FUNCTION_BLOCK FB_SignalLight
VAR_INPUT
	eSafetyState	: E_SafetyState;
	eMachineState 	: E_MachineState;	
END_VAR
VAR_OUTPUT
END_VAR
VAR
	//Blink
	tmrBlink : TON;
	nStateBlink : USINT;
	bBlink	: BOOL;
	
	//Ausgänge für LEDs
	bRed 	AT %Q* : BOOL;
	bYellow AT %Q* : BOOL;
	bGreen	AT %Q* : BOOL;
END_VAR

A_Blink();
IF eSafetyState = E_SafetyState.EmergencyStopPressed THEN
	//rot blinkend
	bRed := TRUE AND bBlink;
	bYellow := FALSE;
	bGreen := FALSE;
	RETURN;
END_IF

CASE eMachineState OF
	E_MachineState.MACHINESTATE_Active, E_MachineState.MACHINESTATE_Running:
		bRed := FALSE;
		bYellow := FALSE;
		bGreen := TRUE;
	E_MachineState.MACHINESTATE_Error:
		bRed := TRUE;
		bYellow := FALSE;
		bGreen := FALSE;		
	E_MachineState.MACHINESTATE_Idle:
		bRed := FALSE;
		bGreen := FALSE;
		IF eSafetyState = E_SafetyState.Locked THEN
			bYellow := TRUE;
		ELSE
			bYellow := TRUE AND bBlink;
		END_IF
	ELSE
		bRed := FALSE;
		bYellow := FALSE;
		bGreen := TRUE AND bBlink;
END_CASE

ACTION A_Blink:
//Phase1
IF nStateBlink = 0 THEN
	bBlink := TRUE;
	tmrBlink(IN:= TRUE, PT:= T#1S);
	IF tmrBlink.Q THEN
		tmrBlink(IN:= FALSE);
		nStateBlink := 1;
	END_IF
END_IF

//Phase2
IF nStateBlink = 1 THEN
	bBlink := FALSE;
	tmrBlink(IN:= TRUE, PT:= T#1S);
	IF tmrBlink.Q THEN
		tmrBlink(IN:= FALSE);
		nStateBlink := 0;
	END_IF
END_IF
END_ACTION

END_FUNCTION_BLOCK

(* stored: Version 1.1.0.1, ProductVersion 3.1.4024.11
   POU FB_SignalLight: Id {e61a5e4c-0cc9-4413-9f08-b41d024678ef}, SpecialFunc None
   Action A_Blink: Id {2ab1c633-f803-4944-8feb-ba268ead02a1} *)
